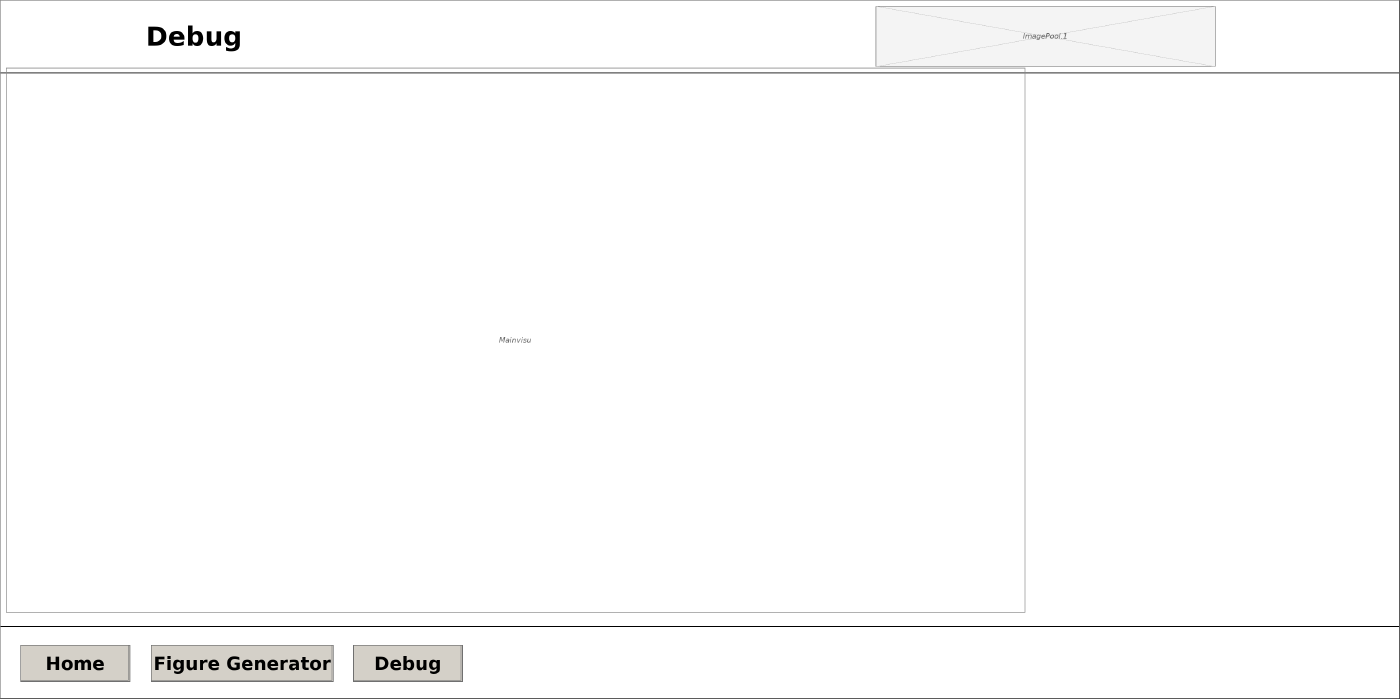
VISUALIZATION Debug  // 1919x959
    Rectangle (0,0 1919x910)
    Rectangle (0,0 1919x100)
    Rectangle (0,859 1919x100)
    Button (28,885 150x50), "Home"
        OnMouseClick: change screen: Home
    Label (191,25 150x50), "Debug"
    Image (1200,8 466x83), image: ImagePool.1
    Button (207,885 250x50), "Figure Generator"
        OnMouseClick: change screen: FigureGenerator1
    Button (484,885 150x50), "Debug"
    Frame (8,93 1397x747)
        shows Mainvisu()
END_VISUALIZATION

(* stored: Version 1.1.0.1, ProductVersion 3.1.4024.12
   Visu Debug: Id {1b0f70c6-0705-4a44-a095-350e20bac033} *)
